// TIA Portal V17 export
// export: Created 2022-02-03T14:45:10.0979599Z, ExportSetting WithDefaults, DisplayName Totally Integrated Automation Portal, DisplayVersion V17, DisplayName TIA Portal Openness, DisplayVersion V17, DisplayName TIA Portal Version Control Interface, DisplayVersion V17, DisplayName SINAMICS Startdrive Advanced, DisplayVersion V17, DisplayName SINAMICS Startdrive G130, G150, S120, S150, SINAMICS MV, S210, DisplayVersion V17, DisplayName SINAMICS Startdrive G110M, G120, G120C, G120D, G120P, G115D, DisplayVersion V17, DisplayName STEP 7 Professional, DisplayVersion V17, DisplayName STEP 7 Safety, DisplayVersion V17, DisplayName WinCC Advanced, DisplayVersion V17
FUNCTION "Mode" : Void   // FC1, LAD
VERSION : 0.1
// stored: Access Unpublished, AutoNumber true, IsIECCheckEnabled false, SetENOAutomatically false, UDAEnableTagReadback false
   VAR_INPUT
      operationAuto : Bool;
      operationManu : Bool;
   END_VAR
   VAR_IN_OUT
      operationMode : Bool;
   END_VAR
BEGIN

REGION Network 1
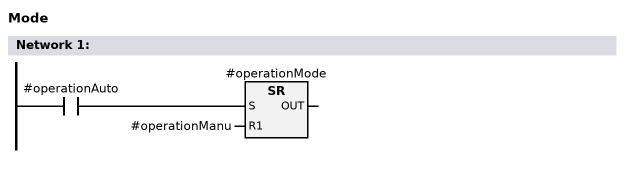
   RUNG wire#powerrail
      Contact( #operationAuto )
      S_SR(operand := #operationMode, r1 := #operationManu)
   END_RUNG
   // the same network as SCL:
   IF #operationAuto THEN
       #operationMode := TRUE;   // SR flip-flop
   END_IF;
   IF #operationManu THEN #operationMode := FALSE; END_IF;
END_REGION
END_FUNCTION
